SUBAPPLICATION Reset_Tageszaehler (* Subapplication Type *)
  (* Standard: 61499-2 *)
  (* Version 1.0, 2023-02-17, Franz *)
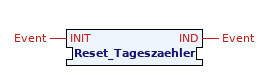
  EVENT_INPUT
    INIT;
  END_EVENT
  EVENT_OUTPUT
    IND;
  END_EVENT
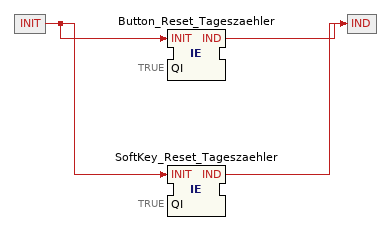
  FBS
    Button_Reset_Tageszaehler : IE(QI := TRUE);
    SoftKey_Reset_Tageszaehler : IE(QI := TRUE);
  END_FBS
  EVENT_CONNECTIONS
    INIT TO Button_Reset_Tageszaehler.INIT;
    Button_Reset_Tageszaehler.IND TO IND;
    INIT TO SoftKey_Reset_Tageszaehler.INIT;
    SoftKey_Reset_Tageszaehler.IND TO IND;
  END_CONNECTIONS
END_SUBAPPLICATION
